RoboDK station: TEMPLATE.rdk

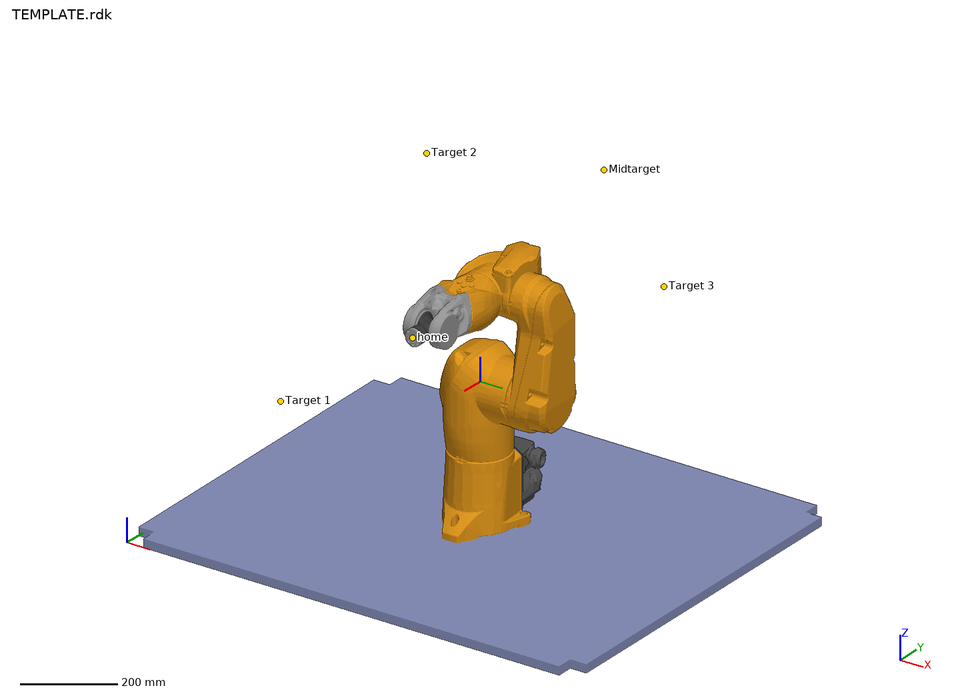
[picture v0: the station drawn from its stored meshes, robots at their saved joint values, targets as dots, program paths as lines]
Station TEMPLATE (saved by RoboDK 5.6.9). Poses are relative to the parent item; angles as X-Y-Z fixed-axis rotations.
  - frame world at (0, 0, 0) mm
    - frame Staubli TX2-40 Base at (560, 460, 340) mm, rotated rx 0 ry 0 rz -90 deg
      - robot Staubli TX2-40: 6 axes, payload 2 kg, reach 515 mm, repeatability 0.02 mm, weight 29 kg
          modified DH rows (alpha deg, a mm, theta deg, d mm): 0, 0, 0, 320; -90, 0, -90, 35; 0, 225, -90, 0; -90, 0, 0, 225; 90, 0, 0, 0; -90, 0, 180, 65
          base shift (0, 0, -320) mm
          joint limits [-180, -125, -138, -270, -120, -270] to [180, 125, 138, 270, 133.5, 270]; home [0, 0, 90, 0, 0, 0]; saved at [0, 0, 90, 0, 0, 0]
    - object Arbeitsflaeche_geteilt at (0, 0, 0) mm, size 1120 x 920 x 20 mm, geometry from Arbeitsflaeche_geteilt.iges
    - object Arbeitsflaeche_komplett at (0, 0, 0) mm, size 1120 x 920 x 20 mm, geometry from Arbeitsflaeche_komplett.IGS
    - object Zelle at (0, 0, 0) mm, rotated rx 90 ry 0 rz -90 deg, size 1120 x 1947.8 x 1200 mm, geometry from Zelle.stp
    - target home (Cartesian target) at (595, 170, 565) mm, rotated rx 0 ry 90 rz -90 deg; joints [0, 0, 90, 0, 0, 0] of Staubli TX2-40
    - target Target 1 (Cartesian target) at (217.63, 235.88, 288.72) mm, rotated rx 180 ry -2.04 rz 54.55 deg; joints [-61.555, 63.778, 48.621, -0.959, 69.437, -25.754] of Staubli TX2-40
    - target Target 2 (Cartesian target) at (302.23, 637.68, 716.85) mm, rotated rx -29.45 ry -2.04 rz 54.55 deg; joints [-132.041, 21.748, 38.604, 170.413, 31.589, -257.058] of Staubli TX2-40
    - target Target 3 (Cartesian target) at (941.54, 573.08, 617.55) mm, rotated rx -94.22 ry -12.46 rz -38.02 deg; joints [-73.787, -42.605, -16.178, 49.565, -48.494, 36.764] of Staubli TX2-40
    - target Midtarget (Cartesian target) at (689.85, 717.16, 755.12) mm, rotated rx -12.87 ry -63.76 rz -90 deg; joints [-21.231, -27.884, -5.338, 11.994, -31.643, -0.983] of Staubli TX2-40
  - Python program Prog1 (listed below)

--- Python program Prog1 ---
# Type help("robodk.robolink") or help("robodk.robomath") for more information
# Press F5 to run the script
# Documentation: https://robodk.com/doc/en/RoboDK-API.html
# Reference:     https://robodk.com/doc/en/PythonAPI/robodk.html
# Note: It is not required to keep a copy of this file, your Python script is saved with your RDK project
from robodk import *      # RoboDK API
from robolink import *    # Robot link toolbox

# Link to RoboDK
RDK = Robolink()

robot = RDK.Item('Staubli TX2-40')

world = RDK.Item('world')
home = RDK.Item('home')
target1 = RDK.Item('Target 1')
target2 = RDK.Item('Target 2')
target3 = RDK.Item('Target 3')
midtarget = RDK.Item('Midtarget')

print('start')

robot.setAccelerationJoints(150)
robot.setSpeedJoints(75)

robot.MoveJ(home)
robot.MoveJ(target1)
robot.MoveJ(target2)
robot.MoveJ(target3)
robot.MoveJ(home)

print('end')
